// TIA Portal V20 export
DATA_BLOCK "500_Hardware"   // DB109
// stored: MemoryReserve 100
   VAR
      Axis : Struct
         MasterVirtual : DB_ANY := 85;
         UnwinderVirtual : DB_ANY := 391;
         UnwinderTop : DB_ANY := 364;
         UnwinderBottom : DB_ANY := 263;
         FinalRoller : DB_ANY := 171;
         Compensator : DB_ANY := 143;
         AnodePnPX1 : DB_ANY := 144;
         AnodePnPX2 : DB_ANY := 145;
         AnodePnPZ1 : DB_ANY := 149;
         AnodePnPZ2 : DB_ANY := 150;
         CathodePnPX1 : DB_ANY := 146;
         CathodePnPX2 : DB_ANY := 147;
         CathodePnPZ1 : DB_ANY := 151;
         CathodePnPZ2 : DB_ANY := 153;
         AnodeMandrelYFront : DB_ANY := 163;
         AnodeMandrelYRear : DB_ANY := 162;
         AnodeMandrelZFront : DB_ANY := 167;
         AnodeMandrelZRear : DB_ANY := 166;
         CathodeMandrelYFront : DB_ANY := 161;
         CathodeMandrelYRear : DB_ANY := 160;
         CathodeMandrelZFront : DB_ANY := 165;
         CathodeMandrelZRear : DB_ANY := 164;
         SepaClampX : DB_ANY := 178;
      END_STRUCT;
      Cam : Struct
         FinalRollerCam { ExternalAccessible := 'False'; ExternalVisible := 'False'; ExternalWritable := 'False'} : DB_ANY := 281;
         CompensatorCam { ExternalAccessible := 'False'; ExternalVisible := 'False'; ExternalWritable := 'False'} : DB_ANY := 69;
         AnodePnPX1Cam { ExternalAccessible := 'False'; ExternalVisible := 'False'; ExternalWritable := 'False'} : DB_ANY := 230;
         AnodePnPX2Cam { ExternalAccessible := 'False'; ExternalVisible := 'False'; ExternalWritable := 'False'} : DB_ANY := 295;
         AnodePnPZ1Cam { ExternalAccessible := 'False'; ExternalVisible := 'False'; ExternalWritable := 'False'} : DB_ANY := 294;
         AnodePnPZ2Cam { ExternalAccessible := 'False'; ExternalVisible := 'False'; ExternalWritable := 'False'} : DB_ANY := 296;
         CathodePnPX1Cam { ExternalAccessible := 'False'; ExternalVisible := 'False'; ExternalWritable := 'False'} : DB_ANY := 293;
         CathodePnPX2Cam { ExternalAccessible := 'False'; ExternalVisible := 'False'; ExternalWritable := 'False'} : DB_ANY := 297;
         CathodePnPZ1Cam { ExternalAccessible := 'False'; ExternalVisible := 'False'; ExternalWritable := 'False'} : DB_ANY := 299;
         CathodePnPZ2Cam { ExternalAccessible := 'False'; ExternalVisible := 'False'; ExternalWritable := 'False'} : DB_ANY := 298;
         AnodeMandrelYFrontCam { ExternalAccessible := 'False'; ExternalVisible := 'False'; ExternalWritable := 'False'} : DB_ANY := 283;
         AnodeMandrelYRearCam { ExternalAccessible := 'False'; ExternalVisible := 'False'; ExternalWritable := 'False'} : DB_ANY := 285;
         AnodeMandrelZFrontCam { ExternalAccessible := 'False'; ExternalVisible := 'False'; ExternalWritable := 'False'} : DB_ANY := 287;
         AnodeMandrelZRearCam { ExternalAccessible := 'False'; ExternalVisible := 'False'; ExternalWritable := 'False'} : DB_ANY := 290;
         CathodeMandrelYFrontCam { ExternalAccessible := 'False'; ExternalVisible := 'False'; ExternalWritable := 'False'} : DB_ANY := 284;
         CathodeMandrelYRearCam { ExternalAccessible := 'False'; ExternalVisible := 'False'; ExternalWritable := 'False'} : DB_ANY := 289;
         CathodeMandrelZFrontCam { ExternalAccessible := 'False'; ExternalVisible := 'False'; ExternalWritable := 'False'} : DB_ANY := 286;
         CathodeMandrelZRearCam { ExternalAccessible := 'False'; ExternalVisible := 'False'; ExternalWritable := 'False'} : DB_ANY := 288;
      END_STRUCT;
      OutputCam : Struct
         FinalRollerXFwdOutputCam { ExternalAccessible := 'False'; ExternalVisible := 'False'; ExternalWritable := 'False'} : DB_ANY := 224;
         FinalRollerXBwdOutputCam { ExternalAccessible := 'False'; ExternalVisible := 'False'; ExternalWritable := 'False'} : DB_ANY := 225;
         FinalRollerXStackTableDownOutputCam { ExternalAccessible := 'False'; ExternalVisible := 'False'; ExternalWritable := 'False'} : DB_ANY := 206;
         FinalRollerXStackAnodeVisionOutputCam { ExternalAccessible := 'False'; ExternalVisible := 'False'; ExternalWritable := 'False'} : DB_ANY := 446;
         FinalRollerXStackCathodeVisionOutputCam { ExternalAccessible := 'False'; ExternalVisible := 'False'; ExternalWritable := 'False'} : DB_ANY := 445;
         AnodePnPX1FwdOutputCam { ExternalAccessible := 'False'; ExternalVisible := 'False'; ExternalWritable := 'False'} : DB_ANY := 413;
         AnodePnPX1BwdOutputCam { ExternalAccessible := 'False'; ExternalVisible := 'False'; ExternalWritable := 'False'} : DB_ANY := 412;
         AnodePnPX2FwdOutputCam { ExternalAccessible := 'False'; ExternalVisible := 'False'; ExternalWritable := 'False'} : DB_ANY := 415;
         AnodePnPX2BwdOutputCam { ExternalAccessible := 'False'; ExternalVisible := 'False'; ExternalWritable := 'False'} : DB_ANY := 414;
         AnodePnPZ1Down1OutputCam { ExternalAccessible := 'False'; ExternalVisible := 'False'; ExternalWritable := 'False'} : DB_ANY := 441;
         AnodePnPZ1Up1OutputCam { ExternalAccessible := 'False'; ExternalVisible := 'False'; ExternalWritable := 'False'} : DB_ANY := 420;
         AnodePnPZ2Down1OutputCam { ExternalAccessible := 'False'; ExternalVisible := 'False'; ExternalWritable := 'False'} : DB_ANY := 437;
         AnodePnPZ2Up1OutputCam { ExternalAccessible := 'False'; ExternalVisible := 'False'; ExternalWritable := 'False'} : DB_ANY := 438;
         AnodePnPZ1Down2OutputCam { ExternalAccessible := 'False'; ExternalVisible := 'False'; ExternalWritable := 'False'} : DB_ANY := 430;
         AnodePnPZ1Up2OutputCam { ExternalAccessible := 'False'; ExternalVisible := 'False'; ExternalWritable := 'False'} : DB_ANY := 432;
         AnodePnPZ2Down2OutputCam { ExternalAccessible := 'False'; ExternalVisible := 'False'; ExternalWritable := 'False'} : DB_ANY := 436;
         AnodePnPZ2Up2OutputCam { ExternalAccessible := 'False'; ExternalVisible := 'False'; ExternalWritable := 'False'} : DB_ANY := 434;
         AnodePnPZ1SuctionOnOutputCam { ExternalAccessible := 'False'; ExternalVisible := 'False'; ExternalWritable := 'False'} : DB_ANY := 433;
         AnodePnPZ1SuctionOffOutputCam { ExternalAccessible := 'False'; ExternalVisible := 'False'; ExternalWritable := 'False'} : DB_ANY := 431;
         AnodePnPZ1ReelCutBlowOutputCam { ExternalAccessible := 'False'; ExternalVisible := 'False'; ExternalWritable := 'False'} : DB_ANY := 185;
         AnodePnPZ2SuctionOnOutputCam { ExternalAccessible := 'False'; ExternalVisible := 'False'; ExternalWritable := 'False'} : DB_ANY := 435;
         AnodePnPZ2SuctionOffOutputCam { ExternalAccessible := 'False'; ExternalVisible := 'False'; ExternalWritable := 'False'} : DB_ANY := 442;
         AnodeAlignSuctionOnOutputCam { ExternalAccessible := 'False'; ExternalVisible := 'False'; ExternalWritable := 'False'} : DB_ANY := 455;
         AnodeAlignSuctionOffOutputCam { ExternalAccessible := 'False'; ExternalVisible := 'False'; ExternalWritable := 'False'} : DB_ANY := 456;
         AnodePnPZ1ReelCutDataDeleteOnOutputCam { ExternalAccessible := 'False'; ExternalVisible := 'False'; ExternalWritable := 'False'} : DB_ANY := 134;
         AnodePnP1XReelCutDataDeleteOffOutputCam { ExternalAccessible := 'False'; ExternalVisible := 'False'; ExternalWritable := 'False'} : DB_ANY := 140;
         AnodeAlignVisionOutputCam { ExternalAccessible := 'False'; ExternalVisible := 'False'; ExternalWritable := 'False'} : DB_ANY := 187;
         CathodePnPX1FwdOutputCam { ExternalAccessible := 'False'; ExternalVisible := 'False'; ExternalWritable := 'False'} : DB_ANY := 417;
         CathodePnPX1BwdOutputCam { ExternalAccessible := 'False'; ExternalVisible := 'False'; ExternalWritable := 'False'} : DB_ANY := 416;
         CathodePnPX2FwdOutputCam { ExternalAccessible := 'False'; ExternalVisible := 'False'; ExternalWritable := 'False'} : DB_ANY := 418;
         CathodePnPX2BwdOutputCam { ExternalAccessible := 'False'; ExternalVisible := 'False'; ExternalWritable := 'False'} : DB_ANY := 419;
         CathodePnPZ1Down1OutputCam { ExternalAccessible := 'False'; ExternalVisible := 'False'; ExternalWritable := 'False'} : DB_ANY := 422;
         CathodePnPZ1Up1OutputCam { ExternalAccessible := 'False'; ExternalVisible := 'False'; ExternalWritable := 'False'} : DB_ANY := 423;
         CathodePnPZ2Down1OutputCam { ExternalAccessible := 'False'; ExternalVisible := 'False'; ExternalWritable := 'False'} : DB_ANY := 428;
         CathodePnPZ2Up1OutputCam { ExternalAccessible := 'False'; ExternalVisible := 'False'; ExternalWritable := 'False'} : DB_ANY := 429;
         CathodePnPZ1Down2OutputCam { ExternalAccessible := 'False'; ExternalVisible := 'False'; ExternalWritable := 'False'} : DB_ANY := 421;
         CathodePnPZ1Up2OutputCam { ExternalAccessible := 'False'; ExternalVisible := 'False'; ExternalWritable := 'False'} : DB_ANY := 439;
         CathodePnPZ2Down2OutputCam { ExternalAccessible := 'False'; ExternalVisible := 'False'; ExternalWritable := 'False'} : DB_ANY := 427;
         CathodePnPZ2Up2OutputCam { ExternalAccessible := 'False'; ExternalVisible := 'False'; ExternalWritable := 'False'} : DB_ANY := 425;
         CathodePnPZ1SuctionOnOutputCam { ExternalAccessible := 'False'; ExternalVisible := 'False'; ExternalWritable := 'False'} : DB_ANY := 457;
         CathodePnPZ1SuctionOffOutputCam { ExternalAccessible := 'False'; ExternalVisible := 'False'; ExternalWritable := 'False'} : DB_ANY := 443;
         CathodePnPZ1ReelCutBlowOutputCam { ExternalAccessible := 'False'; ExternalVisible := 'False'; ExternalWritable := 'False'} : DB_ANY := 424;
         CathodePnPZ2SuctionOnOutputCam { ExternalAccessible := 'False'; ExternalVisible := 'False'; ExternalWritable := 'False'} : DB_ANY := 426;
         CathodePnPZ2SuctionOffOutputCam { ExternalAccessible := 'False'; ExternalVisible := 'False'; ExternalWritable := 'False'} : DB_ANY := 444;
         CathodeAlignSuctionOnOutputCam { ExternalAccessible := 'False'; ExternalVisible := 'False'; ExternalWritable := 'False'} : DB_ANY := 440;
         CathodeAlignSuctionOffOutputCam { ExternalAccessible := 'False'; ExternalVisible := 'False'; ExternalWritable := 'False'} : DB_ANY := 458;
         CathodePnPZ1ReelCutDataDeleteOnOutputCam { ExternalAccessible := 'False'; ExternalVisible := 'False'; ExternalWritable := 'False'} : DB_ANY := 182;
         CathodePnP1XReelCutDataDeleteOffOutputCam { ExternalAccessible := 'False'; ExternalVisible := 'False'; ExternalWritable := 'False'} : DB_ANY := 186;
         CathodeAlignVisionOutputCam { ExternalAccessible := 'False'; ExternalVisible := 'False'; ExternalWritable := 'False'} : DB_ANY := 195;
      END_STRUCT;
   END_VAR
BEGIN
END_DATA_BLOCK
